FUNCTION_BLOCK FB_StartStop
VAR_INPUT
	enable : BOOL;
	reset: BOOL;
	value : REAL;
	StartValue : REAL;
	StopValue : REAL;
	GreaterThan	: BOOL;
	OffDelay	: TIME;
	OnDelay		: TIME;	
END_VAR
VAR_OUTPUT
	Q : BOOL;
END_VAR
VAR
	SR_Started : SR;
	ton_set : TON;
	ton_reset: TON;
	ton_minruntime : TON;
END_VAR

ton_set(PT := Ondelay);
ton_reset(PT := Ondelay);
ton_minruntime(PT := OffDelay);
SR_Started();

IF GreaterThan THEN
	ton_set.IN:= value >= StartValue AND NOT reset;
	ton_reset.IN:= value <= StopValue OR reset;
ELSE
	ton_set.IN:= value <= StartValue AND NOT reset;
	ton_reset.IN:= Value >= StopValue OR reset;
END_IF

ton_minruntime(IN:= sr_started.Q1);
IF enable THEN
	SR_Started.SET1 := ton_set.Q;
	SR_Started.RESET := ton_reset.Q AND ton_minruntime.Q;
	Q := sr_started.Q1;	
ELSE
	SR_Started.SET1 := FALSE;
	SR_Started.RESET := TRUE;
	Q := FALSE;
END_IF

END_FUNCTION_BLOCK

(* stored: Version 1.1.0.1, ProductVersion 3.1.4026.18
   POU FB_StartStop: Id {65b4c91b-4c72-4d6e-85c2-71b432c8e0de}, SpecialFunc None *)
